Staubli VAL3: InterfaceCS8C.pjx

Parameters version=s8.9.1Cs9_BS1830 stackSize=5000 millimeterUnit=true
Program file=screenUpdate.pgx
Program file=start.pgx
Program file=stop.pgx
Data file=InterfaceCS8C.dtx
